RoboDK station: Estacion_Paletizado.rdk

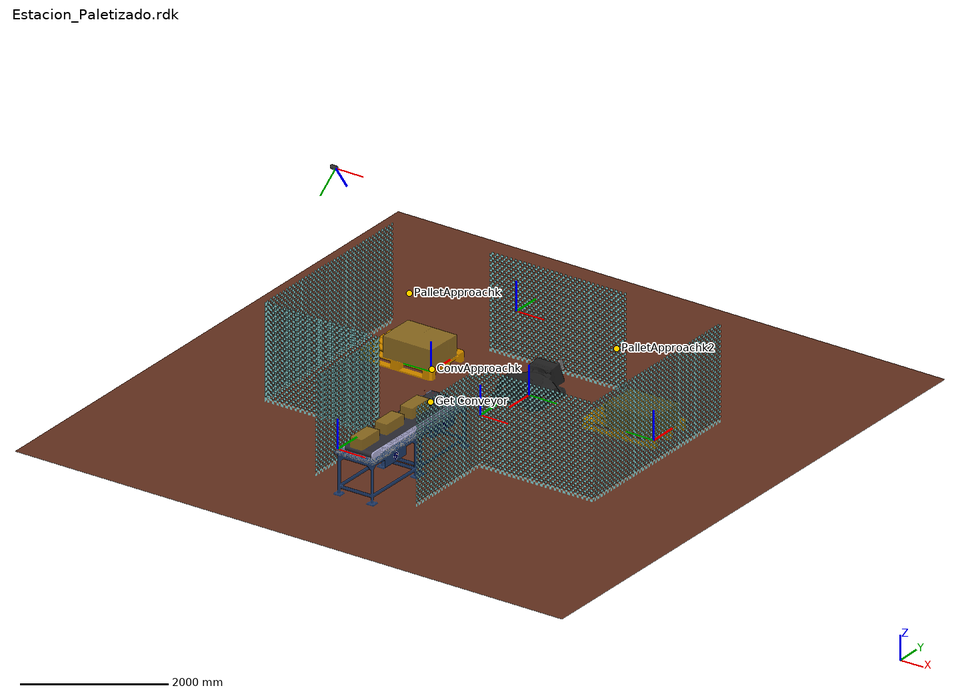
[picture v0: the station drawn from its stored meshes, robots at their saved joint values, targets as dots, program paths as lines]
Station Estacion_Paletizado (saved by RoboDK 5.3.2). Poses are relative to the parent item; angles as X-Y-Z fixed-axis rotations.
Station parameters (name, value as stored): SizeBox, 200, 400, 160, SizePallet, 3,2,2, ConvSpeed, 100.0, SENSOR, 0, parts/min, 2.5, BOX, 84, NBOXP, 12.0, EPALLETE, 1,1, FOTO, 0
  - frame Mundo at (700, 2520, -620) mm
    - object Floor at (0, 0, 0) mm, size 9000 x 9000 x 0 mm, geometry from Floor.sld
    - object Plane 1m x 1m grid at (-725, -2080, 760) mm, rotated rx 0 ry 90 rz 0 deg, size 1500 x 1500 x 0.8 mm, geometry from plane_1m_grid.sld
    - object Plane 1m x 1m grid at (-1850, -1340, 760) mm, rotated rx 0 ry 90 rz 90 deg, size 1500 x 1500 x 0.8 mm, geometry from plane_1m_grid.sld
    - object Plane 1m x 1m grid at (-2600, 910, 750) mm, rotated rx 0 ry 90 rz 0 deg, size 1500 x 1500 x 0.8 mm, geometry from plane_1m_grid.sld
    - object Plane 1m x 1m grid at (-1475, -1340, 760) mm, rotated rx 0 ry 90 rz 90 deg, size 1500 x 1500 x 0.8 mm, geometry from plane_1m_grid.sld
    - object Plane 1m x 1m grid at (-265, 1670, 760) mm, rotated rx 0 ry 90 rz -90 deg, size 1500 x 1500 x 0.8 mm, geometry from plane_1m_grid.sld
    - object Plane 1m x 1m grid at (485, 1670, 760) mm, rotated rx 0 ry 90 rz -90 deg, size 1500 x 1500 x 0.8 mm, geometry from plane_1m_grid.sld
    - object Plane 1m x 1m grid at (2795, 910, 760) mm, rotated rx 0 ry 90 rz -180 deg, size 1500 x 1500 x 0.8 mm, geometry from plane_1m_grid.sld
    - object Plane 1m x 1m grid at (2795, -590, 760) mm, rotated rx 0 ry 90 rz -180 deg, size 1500 x 1500 x 0.8 mm, geometry from plane_1m_grid.sld
    - object Plane 1m x 1m grid at (2040, -1340, 760) mm, rotated rx 0 ry 90 rz 90 deg, size 1500 x 1500 x 0.8 mm, geometry from plane_1m_grid.sld
    - object Plane 1m x 1m grid at (-2600, -590, 760) mm, rotated rx 0 ry 90 rz 0 deg, size 1500 x 1500 x 0.8 mm, geometry from plane_1m_grid.sld
    - object Plane 1m x 1m grid at (1665, -1340, 760) mm, rotated rx 0 ry 90 rz 90 deg, size 1500 x 1500 x 0.8 mm, geometry from plane_1m_grid.sld
    - object Plane 1m x 1m grid at (925, -2080, 760) mm, rotated rx 0 ry 90 rz 0 deg, size 1500 x 1500 x 0.8 mm, geometry from plane_1m_grid.sld
    - object Table 1400x800x800 at (110, -1140, 645) mm, rotated rx 0 ry 0 rz -90 deg, size 1138.7 x 657.6 x 641.5 mm, geometry from Table-1400mmx800mmx800mm.sld
    - object Table 1400x800x800 at (110, -2280, 645) mm, rotated rx 0 ry 0 rz -90 deg, size 1138.7 x 657.6 x 641.5 mm, geometry from Table-1400mmx800mmx800mm.sld
  - frame KR Base at (900, 3380, -610) mm, rotated rx 0 ry 0 rz -90 deg
    - robot KR (model KUKA KR 120 R3200 PA): 4 axes, payload 120 kg, reach 3195 mm, repeatability 0.06 mm, weight 1075 kg
        joint limits [-185, -140, 0, -350] to [185, -5, 155, 350]; home [0, -100.15, 95.16, -180.59]; saved at [80.379, -89.016, 111.792, -188.281]
      - tool GripperK, TCP at (0, 0, 80) mm, rotated rx 0 ry 0 rz 90 deg, size 461.9 x 92.4 x 220 mm, geometry from test.iges
      - tool TCPK, TCP at (0, 0, 160) mm, rotated rx 0 ry 0 rz 90 deg
    - target ConvApproachk (joint target) at (2164.54, -72.94, 1237.21) mm, rotated rx -180 ry 0 rz -90.59 deg; joints [1.93, -73.65, 92.328, -178.66, 0, 0] of KR
    - target PalletApproachk (joint target) at (297.16, -1753.05, 1156.5) mm, rotated rx 180 ry 0 rz -178.66 deg; joints [80.379, -89.016, 111.792, -188.281, 0, 0] of KR
    - target PalletApproachk2 (joint target) at (316.59, 1666.46, 1294.36) mm, rotated rx 180 ry 0 rz -180 deg; joints [-79.243, -94.763, 109.774, 10.757] of KR
    - frame PalletK2 at (419.96, 2346.44, 151.5) mm, rotated rx 0 ry 0 rz 180 deg
      - object EuropalletK at (0, 0, 0) mm, size 800 x 144 x 1200 mm, geometry from User Library-Europallet.igs
      - object Part at (100.16, 200.94, 79.97) mm, rotated rx 0 ry 0 rz -180 deg, size 200 x 400 x 160 mm, geometry from box.sld
      - object Part at (300.16, 202.94, 79.97) mm, rotated rx 0 ry 0 rz -180 deg, size 200 x 400 x 160 mm, geometry from box.sld
      - object Part at (500.16, 199.94, 79.97) mm, rotated rx 0 ry 0 rz 180 deg, size 200 x 400 x 160 mm, geometry from box.sld
      - object Part at (100.16, 579.94, 79.97) mm, rotated rx 0 ry 0 rz 180 deg, size 200 x 400 x 160 mm, geometry from box.sld
      - object Part at (300.16, 601.94, 79.97) mm, rotated rx 0 ry 0 rz 180 deg, size 200 x 400 x 160 mm, geometry from box.sld
      - object Part at (500.16, 600.94, 79.97) mm, rotated rx 0 ry 0 rz -180 deg, size 200 x 400 x 160 mm, geometry from box.sld
      - object Part at (100.16, 199.94, 239.97) mm, rotated rx 0 ry 0 rz 180 deg, size 200 x 400 x 160 mm, geometry from box.sld
      - object Part at (300.16, 202.94, 239.97) mm, rotated rx 0 ry 0 rz 180 deg, size 200 x 400 x 160 mm, geometry from box.sld
      - object Part at (500.16, 202.94, 239.97) mm, rotated rx 0 ry 0 rz -180 deg, size 200 x 400 x 160 mm, geometry from box.sld
      - object Part at (100.16, 602.94, 239.97) mm, rotated rx 0 ry 0 rz -180 deg, size 200 x 400 x 160 mm, geometry from box.sld
      - object Part at (300.16, 607.94, 239.97) mm, rotated rx 0 ry 0 rz -180 deg, size 200 x 400 x 160 mm, geometry from box.sld
      - object Part at (500.16, 598.94, 239.97) mm, rotated rx 0 ry 0 rz 180 deg, size 200 x 400 x 160 mm, geometry from box.sld
    - frame PalletK at (419.96, -1313.56, 151.5) mm, rotated rx 0 ry 0 rz 180 deg
      - object EuropalletK at (0, 0, 0) mm, size 800 x 144 x 1200 mm, geometry from User Library-Europallet.igs
      - object Part at (100.16, 203.94, 79.97) mm, rotated rx 0 ry 0 rz 180 deg, size 200 x 400 x 160 mm, geometry from box.sld
      - object Part at (300.16, 202.94, 79.97) mm, rotated rx 0 ry 0 rz -180 deg, size 200 x 400 x 160 mm, geometry from box.sld
      - object Part at (500.16, 202.94, 79.97) mm, rotated rx 0 ry 0 rz 180 deg, size 200 x 400 x 160 mm, geometry from box.sld
      - object Part at (100.16, 596.94, 79.97) mm, rotated rx 0 ry 0 rz -180 deg, size 200 x 400 x 160 mm, geometry from box.sld
      - object Part at (300.16, 602.94, 79.97) mm, rotated rx 0 ry 0 rz -180 deg, size 200 x 400 x 160 mm, geometry from box.sld
      - object Part at (500.16, 603.94, 79.97) mm, rotated rx 0 ry 0 rz 180 deg, size 200 x 400 x 160 mm, geometry from box.sld
      - object Part at (100.16, 201.94, 239.97) mm, rotated rx 0 ry 0 rz -180 deg, size 200 x 400 x 160 mm, geometry from box.sld
      - object Part at (300.16, 201.94, 239.97) mm, rotated rx 0 ry 0 rz 180 deg, size 200 x 400 x 160 mm, geometry from box.sld
      - object Part at (500.16, 194.94, 239.97) mm, rotated rx 0 ry 0 rz 180 deg, size 200 x 400 x 160 mm, geometry from box.sld
      - object Part at (100.16, 596.94, 239.97) mm, rotated rx 0 ry 0 rz 180 deg, size 200 x 400 x 160 mm, geometry from box.sld
      - object Part at (300.16, 602.94, 239.97) mm, rotated rx 0 ry 0 rz 180 deg, size 200 x 400 x 160 mm, geometry from box.sld
      - object Part at (500.16, 599.94, 239.97) mm, rotated rx 0 ry 0 rz -180 deg, size 200 x 400 x 160 mm, geometry from box.sld
  - frame ConveyorReference at (597.23, -679.82, 119.18) mm
    - robot Conveyor Belt: 1 axes
        modified DH rows (alpha deg, a mm, theta deg, d mm): 0, 0, 0, 0 linear
        base shift (440, 200, 0) mm, rotated rx 0 ry 90 rz 90 deg
        joint limits [-500000] to [500000]; home [0]; saved at [50536]
      - frame MovingRef at (0, 0, 0) mm
        - object Part at (-49217, 240, 80) mm, rotated rx 0 ry 0 rz -90 deg, size 200 x 400 x 160 mm, geometry from box.sld
        - object Part at (-49811, 240, 80) mm, rotated rx 0 ry 0 rz -90 deg, size 200 x 400 x 160 mm, geometry from box.sld
        - object Part at (-50391, 240, 80) mm, rotated rx 0 ry 0 rz -90 deg, size 200 x 400 x 160 mm, geometry from box.sld
    - object box100mm at (200, 300, 0) mm, size 100 x 100 x 100 mm, geometry from box.sld
    - object Sensor SICK WL4S at (551.19, 2078.29, 24.16) mm, rotated rx 90 ry 0 rz 180 deg, size 683.3 x 45.2 x 12.5 mm, geometry from SICK WL4S-3P1330-Order no.1042068 (1).stp
      - Python program SensorActivate (listed below)
    - target Get Conveyor (Cartesian target) at (200.16, 1899.94, 0.03) mm, rotated rx -180 ry 0 rz -180 deg; joints [2.72, -64.765, 103.115, -177.28, 0, 0] of KR
  - frame Camera Reference at (780, -980, 4500) mm, rotated rx -145 ry 0 rz 0 deg
    - object SICK VSPP-5f2113 at (0, 0, 0) mm, size 53 x 116 x 38 mm, geometry from Cam2D_SICK_VSPP_5F2113.sld
  - Python program SetSimulationParams (listed below)
  - Python program BorradoA (listed below)
  - Python program BorradoB (listed below)
  - Python program AddPart (listed below)
  - Python program InputParts (listed below)
  - Python program RobotPackParts (listed below)
  - Python program Telegram (listed below)
  - Python program Camara (listed below)
  - program MainSimulation (5 instructions, listed below)
  - frame Fajardo_Jacho at (0, 4380, 0) mm

--- Python program SensorActivate ---
# Type help("robolink") or help("robodk") for more information
# Press F5 to run the script
# Note: you do not need to keep a copy of this file, your python script is saved with the station
from robolink import *    # API to communicate with RoboDK
from robodk import *      # basic matrix operations
RDK = Robolink()

# This script allows to simulate a laser sensor
# that detect the presence of a part in a plane,
# such as a part crossing a laser sensor in a
# conveyor belt

# Use a target from the station as a reference plane:
SENSOR_NAME = 'Sensor SICK WL4S'
SENSOR_VARIABLE = 'SENSOR'

# Look for parts with the keyword "Part"
OBJECTS_REFERENCE = 'MovingRef'
moving_ref = RDK.Item(OBJECTS_REFERENCE, ITEM_TYPE_FRAME)

# Update status every 1 ms
RECHECK_PERIOD = 0.001

# Get the sensor and the detection plane
SENSOR = RDK.Item(SENSOR_NAME, ITEM_TYPE_OBJECT)

# Start delayed as some parts may be deleted
pause(2)

# Loop forever to detect parts
detected_status = -1
while True:
    detected = 0
    for obj in moving_ref.Childs():
        # check if an object has the part keyword and is detected by the laser
        if SENSOR.Collision(obj) > 0:
            detected = 1
            break

    # update the current status of the sensor
    if detected_status != detected:
        detected_status = detected
        RDK.setParam(SENSOR_VARIABLE, detected_status)
        print('Object detected status --> %i' % detected_status)

    ESTADOS_PALLET      = RDK.getParam('EPALLETE')
    ESTADOS_PALLET_AB   = [int(x.replace(' ','')) for x in ESTADOS_PALLET.split(',')]
    numero_disponible   = ESTADOS_PALLET_AB[0] + ESTADOS_PALLET_AB[1]

    if numero_disponible == 2:
        # Se detiene el sensor hasta que haya palletes disponibles
        while numero_disponible == 2:
            ESTADOS_PALLET      = RDK.getParam('EPALLETE')
            ESTADOS_PALLET_AB   = [int(x.replace(' ','')) for x in ESTADOS_PALLET.split(',')]
            numero_disponible   = ESTADOS_PALLET_AB[0] + ESTADOS_PALLET_AB[1]
        pause(2)
    # Wait some time...
    pause(RECHECK_PERIOD)

--- Python program SetSimulationParams ---
# Type help("robolink") or help("robodk") for more information
# Press F5 to run the script
# Note: you do not need to keep a copy of this file, your python script is saved with the station
from robolink import *    # API to communicate with RoboDK
from robodk import *      # basic matrix operations

RDK = Robolink()

# Parametros creados en la estacion de trabajo
PARAM_SIZE_BOX = 'SizeBox'
PARAM_SIZE_PALLET = 'SizePallet'
PARAM_CONV_SPEED_MM = 'ConvSpeed'
PARAM_PARTS_X_MINUTE = 'parts/min'

#Valores de los parametros creados en la estacion de trabajo
size_box = RDK.getParam(PARAM_SIZE_BOX)
size_pallet = RDK.getParam(PARAM_SIZE_PALLET)
conv_speed = RDK.getParam(PARAM_CONV_SPEED_MM)
parts_x_minute = RDK.getParam(PARAM_PARTS_X_MINUTE)

# ------------------------------------------------------------
size_box_input = mbox('Enter the size of the box in mm [L,W,H]', entry=size_box)
if size_box_input:
    RDK.setParam(PARAM_SIZE_BOX, size_box_input)
else:
    quit()

# ------------------------------------------------------------
size_pallet_input = mbox('Enter the size of the pallet', entry=size_pallet)
if size_pallet_input:
    RDK.setParam(PARAM_SIZE_PALLET, size_pallet_input)
else:
    quit()


# ------------------------------------------------------------
parts_x_minute_entry = mbox('Enter the number of parts per minute', entry=parts_x_minute)
if parts_x_minute_entry:
    RDK.setParam(PARAM_PARTS_X_MINUTE, parts_x_minute_entry)
else:
    quit()

# ------------------------------------------------------------
conv_speed_input = mbox('Enter the speed of the conveyor in mm/s', entry=conv_speed)
if conv_speed_input:
    RDK.setParam(PARAM_CONV_SPEED_MM, conv_speed_input)
    conv_speed = float(conv_speed_input)
    conv = RDK.Item('Conveyor Belt', ITEM_TYPE_ROBOT)
    conv.setSpeed(conv_speed)

else:
    quit()

--- Python program BorradoA ---
# Type help("robolink") or help("robodk") for more information
# Press F5 to run the script
# Documentation: https://robodk.com/doc/en/RoboDK-API.html
# Reference:     https://robodk.com/doc/en/PythonAPI/index.html
# Note: It is not required to keep a copy of this file, your python script is saved with the station
from robolink import *    # RoboDK API
from robodk import *      # Robot toolbox
RDK = Robolink()

# Variable con la referencia del pallete a borrar
pallete_ref = RDK.Item('PalletK', ITEM_TYPE_FRAME)

#Eliminar las cajas del PalleteA
for obj in pallete_ref.Childs():
    if obj.Name().startswith("Part"):
        obj.Delete()

# Actualizar el estado de palleteA en el parametro EPALLETE
estado_pallete = RDK.getParam('EPALLETE')
l = list(estado_pallete) #El parametro es un string
l[0] = '0'
estado_pallete = "".join(l)
RDK.setParam('EPALLETE', estado_pallete)

--- Python program BorradoB ---
# Type help("robolink") or help("robodk") for more information
# Press F5 to run the script
# Documentation: https://robodk.com/doc/en/RoboDK-API.html
# Reference:     https://robodk.com/doc/en/PythonAPI/index.html
# Note: It is not required to keep a copy of this file, your python script is saved with the station
from robolink import *    # RoboDK API
from robodk import *      # Robot toolbox
RDK = Robolink()

# Variable con la referencia del pallete a borrar
pallete_ref = RDK.Item('PalletK2', ITEM_TYPE_FRAME)

#Eliminar las cqjas del PalleteB
for obj in pallete_ref.Childs():
    if obj.Name().startswith("Part"):
        obj.Delete()

# Actualizar el estado de palleteB en el parametro EPALLETE
estado_pallete = RDK.getParam('EPALLETE')
l = list(estado_pallete) #El parametro es un string
l[2] = '0'
estado_pallete = "".join(l)
RDK.setParam('EPALLETE', estado_pallete)

--- Python program AddPart ---
# Type help("robolink") or help("robodk") for more information
# Press F5 to run the script
# Note: you do not need to keep a copy of this file, your python script is saved with the station
from robolink import *    # API to communicate with RoboDK
from robodk import *      # basic matrix operations
import random
RDK = Robolink()

#Variables con nombre de objeto y referencia a usar
PART_NAME       = 'box100mm'
CONVEYOR_REF    = 'MovingRef'

#Valores de las dimensiones de la caja
SIZE_BOX = RDK.getParam('SizeBox')
SIZE_BOX_XYZ = [float(x.replace(' ','')) for x in SIZE_BOX.split(',')]
[SIZE_BOX_X, SIZE_BOX_Y, SIZE_BOX_Z] = SIZE_BOX_XYZ

# Creacion de nueva caja en la banda
part = RDK.Item(PART_NAME, ITEM_TYPE_OBJECT)
conveyor_ref = RDK.Item(CONVEYOR_REF, ITEM_TYPE_FRAME) #Referencia movil de la banda transportadora
part_pos = part.PoseAbs() # Posicion absoluta de la caja de referencia
part.Copy()
newpart = conveyor_ref.Paste()
newpart.setPoseAbs(part_pos*transl(0,0,SIZE_BOX_Z/2)) #Posicionando la nueva caja teniendo en cuenta su referencia central.
newpart.setName('Part') # Se crea una caja para el palleteA
newpart.Scale([SIZE_BOX_X/100, SIZE_BOX_Y/100, SIZE_BOX_Z/100]) #Escala con respecto al objeto de referencia (100mm cube)
newpart.Recolor([0.678, 0.529, 0.2, 1]) #set RGBA color
newpart.setVisible(True, False) #make item visible but hide the reference frame

--- Python program InputParts ---
# Type help("robolink") or help("robodk") for more information
# Press F5 to run the script
# Note: you do not need to keep a copy of this file, your python script is saved with the station
from robolink import *    # API to communicate with RoboDK
from robodk import *      # basic matrix operations

# Use RoboDK API as RDK
RDK = Robolink()

# Parametros de la estacion
PARAM_PARTS_X_MINUTE = 'parts/min'
PARAM_NUMERO_BOX_PALLETE = 'NBOXP'
PARAM_ESTADO_PALLETE = 'EPALLETE'

# Establecer en 0 el estado de los pallete A y B
RDK.setParam(PARAM_ESTADO_PALLETE, '0,0')

# Establecer el numero indicador de cajas por Pallete
SIZE_PALLET = RDK.getParam('SizePallet')
SIZE_PALLET_XYZ = [float(x.replace(' ','')) for x in SIZE_PALLET.split(',')]
numero_box_pallete = SIZE_PALLET_XYZ[0]*SIZE_PALLET_XYZ[1]*SIZE_PALLET_XYZ[2]
RDK.setParam(PARAM_NUMERO_BOX_PALLETE, numero_box_pallete)

# turn off rendering (much faster when setting up the station)
#RDK.Render(False)

# Eliminar todas las cajas previamente simuladas
all_objects     = RDK.ItemList(ITEM_TYPE_OBJECT, False)
for item in all_objects:
    if item.Name().startswith("Part"):
        item.Delete()

# Turn on rendering
#RDK.Render(True)

# Valor de la cantidad de cajas por minuto
parts_x_minute = RDK.getParam(PARAM_PARTS_X_MINUTE)

# Seleccion del codigo de AddPart
add_part = RDK.Item('AddPart', ITEM_TYPE_PROGRAM_PYTHON)

# Movimiento de la banda transportadora
conv = RDK.Item('Conveyor Belt', ITEM_TYPE_ROBOT)
conv.setJoints([0]) # Establecer en cero
conv.MoveJ([99999], False) # Mover hasta el maximo valor permitido.

# Temporizador para creacion de cajas
SECONDS_X_PART = 60.0 / parts_x_minute #Tiempo por cada caja
tic() # Marcar inicio de cconteo
timer_last = toc() # Tiempo transcurrido desde el inicio del conteo
simulation_time = SECONDS_X_PART
while True:

    # Numero indicador de disponibilidad de pallete
    ESTADOS_PALLET      = RDK.getParam(PARAM_ESTADO_PALLETE)
    ESTADOS_PALLET_AB   = [int(x.replace(' ','')) for x in ESTADOS_PALLET.split(',')]
    numero_disponible   = ESTADOS_PALLET_AB[0] + ESTADOS_PALLET_AB[1]

    # Creacion de la nueva caja
    timer = toc()
    simulation_time = simulation_time + (timer - timer_last) * RDK.SimulationSpeed()
    timer_last = timer
    if simulation_time >= SECONDS_X_PART and numero_disponible != 2: # Se crea mas cajas siempre que haya disponibles un pallete
        simulation_time = simulation_time - SECONDS_X_PART
        add_part.RunProgram()
    if numero_disponible == 2: # No hay disponible pallete
        conv.Stop()
        while numero_disponible == 2: #Espera hasta este disponible el palleteA
            ESTADOS_PALLET      = RDK.getParam(PARAM_ESTADO_PALLETE)
            ESTADOS_PALLET_AB   = [int(x.replace(' ','')) for x in ESTADOS_PALLET.split(',')]
            numero_disponible   = ESTADOS_PALLET_AB[0] + ESTADOS_PALLET_AB[1]
        conv.MoveJ([99999], False)
        tic() # Se reinicia la cuenta para las cajas
        timer_last = toc()
        simulation_time = 0

    pause(0.01)

--- Python program RobotPackParts ---
# Type help("robolink") or help("robodk") for more information
# Press F5 to run the script
# Note: you do not need to keep a copy of this file, your python script is saved with the station
from robolink import *    # API to communicate with RoboDK
from robodk import *      # basic matrix operations

# Use RoboDK API as RL
RDK = Robolink()

# define default approach distance
APPROACH = 100

# Parametros de la estacion
SENSOR_VARIABLE = 'SENSOR'
PARAM_ESTADO_PALLETE = 'EPALLETE'
RDK.setParam(PARAM_ESTADO_PALLETE, '0,0')
ESTADOS_PALLET      = RDK.getParam(PARAM_ESTADO_PALLETE)

# gather robot, tool and reference frames from the station
robot               = RDK.Item('KR', ITEM_TYPE_ROBOT)
tool                = RDK.Item('GripperK', ITEM_TYPE_TOOL)
tool_tcp            = RDK.Item('TCPK', ITEM_TYPE_TOOL)

frame_palletA        = RDK.Item('PalletK', ITEM_TYPE_FRAME)
frame_palletB       = RDK.Item('PalletK2', ITEM_TYPE_FRAME)
frame_conv          = RDK.Item('ConveyorReference', ITEM_TYPE_FRAME)
frame_conv_moving   = RDK.Item('MovingRef', ITEM_TYPE_FRAME)

# gather targets
target_pallet_safeA  = RDK.Item('PalletApproachk', ITEM_TYPE_TARGET)
target_pallet_safeB = RDK.Item('PalletApproachk2', ITEM_TYPE_TARGET)
target_conv_safe    = RDK.Item('ConvApproachk', ITEM_TYPE_TARGET)
target_conv         = RDK.Item('Get Conveyor', ITEM_TYPE_TARGET)

# Reinicio de la cuenta de las cajas totales paletizadas
COUNT_BOX = 0

# get variable parameters
SIZE_BOX = RDK.getParam('SizeBox')
SIZE_PALLET = RDK.getParam('SizePallet')
SIZE_BOX_XYZ = [float(x.replace(' ','')) for x in SIZE_BOX.split(',')]
SIZE_PALLET_XYZ = [float(x.replace(' ','')) for x in SIZE_PALLET.split(',')]
SIZE_BOX_Z = SIZE_BOX_XYZ[2] # the height of the boxes is important to take into account when approaching the positions

def box_calc(size_xyz, pallet_xyz):
    """Calculates a list of points to store parts in a pallet"""
    [size_x, size_y, size_z] = size_xyz
    [pallet_x, pallet_y, pallet_z] = pallet_xyz
    xyz_list = []
    for h in range(int(pallet_z)):
        for j in range(int(pallet_y)):
            for i in range(int(pallet_x)):
                xyz_list = xyz_list + [[(i+0.5)*size_x, (j+0.5)*size_y, (h+0.5)*size_z]]
    return xyz_list

def TCP_On(toolitem):
    """Attaches the closest object to the toolitem Htool pose,
    It will also output appropriate function calls on the generated robot program (call to TCP_On)"""
    toolitem.AttachClosest()
    toolitem.RDK().RunMessage('Set air valve on')
    toolitem.RDK().RunProgram('TCP_On()')

def TCP_Off(toolitem, itemleave=0):
    """Detaches the closest object attached to the toolitem Htool pose,
    It will also output appropriate function calls on the generated robot program (call to TCP_Off)"""
    #toolitem.DetachClosest(itemleave)
    toolitem.DetachAll(itemleave)
    toolitem.RDK().RunMessage('Set air valve off')
    toolitem.RDK().RunProgram('TCP_Off()')

# calculate an array of positions to get/store the parts
parts_positions = box_calc(SIZE_BOX_XYZ, SIZE_PALLET_XYZ)

# Calculate a new TCP that takes into account the size of the part (targets are set to the center of the box)
tool_xyzrpw = tool.PoseTool()*transl(0,0,SIZE_BOX_Z/2)
tool_tcp.setPoseTool(tool_xyzrpw)
#tool_tcp = robot.AddTool(tool_xyzrpw, 'TCP')

# ---------------------------------------------------------------------------------
# -------------------------- PROGRAM START ----------------------------------------

def WaitSensor():
    if RDK.RunMode() == RUNMODE_SIMULATE:
        # Simulate the sensor by waiting for the SENSOR status to turn to 1 (object present)
        while RDK.getParam(SENSOR_VARIABLE) == 0:
            pause(0.001)
    else:
        RDK.RunProgram('WaitSensor')
    print("Part detected")

P = -1 # Variable indicadora del pallete a llenar
robot.setTool(tool_tcp)
nparts = len(parts_positions)
while True:
    # Numero indicador de disponibilidad de palletes
    ESTADOS_PALLET_AB   = [int(x.replace(' ','')) for x in ESTADOS_PALLET.split(',')]
    numero_disponible   = ESTADOS_PALLET_AB[0] + ESTADOS_PALLET_AB[1]

    if numero_disponible == 2:
        # Se detiene el brazo robotico hasta que haya palletes disponibles
        while numero_disponible == 2:
            ESTADOS_PALLET      = RDK.getParam(PARAM_ESTADO_PALLETE)
            ESTADOS_PALLET_AB   = [int(x.replace(' ','')) for x in ESTADOS_PALLET.split(',')]
            numero_disponible   = ESTADOS_PALLET_AB[0] + ESTADOS_PALLET_AB[1]
    #Establecer la referencia y el target del pallete
    if ESTADOS_PALLET_AB[0] == 0:
        P = 1
        frame_pallet = frame_palletA
        target_pallet_safe = target_pallet_safeA
    elif ESTADOS_PALLET_AB[1] == 0:
        P = 2
        frame_pallet = frame_palletB
        target_pallet_safe = target_pallet_safeB

    i = 0
    while i < nparts:
        # ----------- place the box i on the convegor ------
        # approach to the conveyor
        robot.setFrame(frame_conv)
        target_conv_pose = target_conv.Pose()*transl(0,0,-SIZE_BOX_Z/2)
        target_conv_app = target_conv_pose*transl(0,0,-APPROACH)
        robot.MoveJ(target_conv_safe)
        robot.MoveJ(target_conv_app)
        WaitSensor()
        robot.MoveL(target_conv_pose)
        TCP_On(tool) # detach an place the object in the moving reference frame of the conveyor
        robot.MoveL(target_conv_app)
        robot.MoveJ(target_conv_safe)

        # ----------- take a part from the conveyor ------
        # get the xyz position of part i
        robot.setFrame(frame_pallet)
        part_position_i = parts_positions[i]
        target_i = transl(part_position_i)*rotx(pi)
        target_i_app = target_i * transl(0,0,-(APPROACH+SIZE_BOX_Z))
        # approach to the pallet
        robot.MoveJ(target_pallet_safe)
        # get the box i
        robot.MoveJ(target_i_app)
        robot.MoveL(target_i)
        TCP_Off(tool, frame_pallet) # attach the closest part
        robot.MoveL(target_i_app)
        robot.MoveJ(target_pallet_safe)
        COUNT_BOX +=1 # Aumenta la cuenta cuando deja una caja
        RDK.setParam('BOX', COUNT_BOX)
        i = i + 1

    # Cambio del estado de los pallete
    ESTADOS_PALLET      = RDK.getParam(PARAM_ESTADO_PALLETE)
    if P == 1:
        l = list(ESTADOS_PALLET)
        l[0] = '1'
        ESTADOS_PALLET = "".join(l)
    else:
        l = list(ESTADOS_PALLET)
        l[2] = '1'
        ESTADOS_PALLET = "".join(l)
    RDK.setParam('EPALLETE', ESTADOS_PALLET)

--- Python program Telegram ---
#!/usr/bin/env python
# pylint: disable=C0116,W0613
# This program is dedicated to the public domain under the CC0 license.

import logging

from telegram import Update, ForceReply
from telegram.ext import Updater, CommandHandler, MessageHandler, Filters, CallbackContext
from telegram import ChatAction

# Enable logging
logging.basicConfig(
    format='%(asctime)s - %(name)s - %(levelname)s - %(message)s', level=logging.INFO
)

logger = logging.getLogger(__name__)


from robolink import *    # RoboDK API
from robodk import *      # Robot toolbox

RDK = Robolink()
FOTO_ESTACION = 'FOTO' # Parametro que indica si se debe tomar una foto
path_rdk = RDK.getParam('PATH_OPENSTATION')# Parametro con la direccion de la foto
file_name = '/estacion.jpg'# Parametro con el nombre de la foto

# Definiendo los comandos de telegram
def start(update: Update, context: CallbackContext) -> None:
    user = update.effective_user
    update.message.reply_markdown_v2( #Funcion para enviar un mensaje con el nombre del usuario.
        fr'Hola {user.mention_markdown_v2()}\!',
        reply_markup=ForceReply(selective=True),
    )
    update.message.reply_text('En esta aplicacion podras consultar el estado de la estacion de paletizado, usa el comando /help para conocer las funciones')

def help_command(update: Update, context: CallbackContext) -> None:
    update.message.reply_text('Las funciones que se pueden usar son:') # Funcion para enviar un mensaje de texto al usuario
    update.message.reply_text('/help -> Te ayuda a conocer la funciones existentes')
    update.message.reply_text('/box -> Te indica la cantidas de cajas paletizadas')
    update.message.reply_text('/pallete -> Te indica la cantidad de palletes llenos')
    update.message.reply_text('/Epallete -> Te indica el estado de los palletes de la estacion')
    update.message.reply_text('/foto -> Te envia una foto de la estacion')

def echo(update: Update, context: CallbackContext) -> None:
    update.message.reply_text('Por favor, ingrese un comando conocido, o de clic en -> /help')

def box(update: Update, context: CallbackContext) -> None:
    cantidad_cajas = RDK.getParam('BOX') # Parametro con el valor de cajas totales paletizadas
    update.message.reply_text('La cantidad de cajas paletizadas es de ' + str(cantidad_cajas))

def pallete(update: Update, context: CallbackContext) -> None:
    cantidad_cajas = int(RDK.getParam('BOX')) # Parametro con el valor de cajas totales paletizadas
    numero_box_pallete = int(RDK.getParam('NBOXP')) #Parametro con la cantidad de cajas por palleto
    cantidad_pallete = cantidad_cajas//numero_box_pallete # Numero de palletes enteros realizados
    update.message.reply_text('La cantidad de palletes terminados es de ' + str(cantidad_pallete))

def Epallete(update: Update, context: CallbackContext) -> None:
    estado_pallete      = RDK.getParam('EPALLETE') #Parametro con el estado de los palletes
    estados_pallete_AB   = [int(x.replace(' ','')) for x in estado_pallete.split(',')]
    # Asignacion de vacio o lleno al mensaje sobre el estado de cada pallete
    if estados_pallete_AB[0] == 0 :
        palleteA = 'vacio o llenando'
    else:
        palleteA = 'lleno'
    if estados_pallete_AB[1] == 0:
        palleteB = 'vacio o llenando'
    else:
        palleteB = 'lleno'

    # Determinar estructura del mensaje segun el estado de los palletes
    if estados_pallete_AB == [1,1]:
        update.message.reply_text('Los dos palletes se encuentran llenos, el proceso esta detenido' )
    else:
        update.message.reply_text('El palleteA esta ' + str(palleteA))
        update.message.reply_text('El palleteB esta ' + str(palleteB))

def foto(chat):
    chat.send_action(action=ChatAction.UPLOAD_PHOTO,timeout=None) #Accion de que se esta enviando una foto
    pause(0.1)
    chat.send_photo(photo = open(path_rdk+file_name,'rb')) # Se envia la foto que sera buscada en la direccion establecida
    RDK.setParam(FOTO_ESTACION,'0') # Actualizacion de parametro que indica cuando tomar una foto

def chat(update: Update, context: CallbackContext) -> None:
    RDK.setParam(FOTO_ESTACION,'1') # Actualizacion de parametro que indica cuando tomar una foto
    chat = update.message.chat #Datos de chat de la persona que escribe
    foto(chat) # Funcion para enviar la foto

def main() -> None:
    """Start the bot."""
    # Create the Updater and pass it your bot's token.
    updater = Updater("5062967228:AAGSuI74jk8Jqe0g8b1kAKCBIIlwF6qlM4A")

    # Get the dispatcher to register handlers
    dispatcher = updater.dispatcher

    # on different commands - answer in Telegram
    dispatcher.add_handler(CommandHandler("start", start))
    dispatcher.add_handler(CommandHandler("help", help_command))
    dispatcher.add_handler(CommandHandler("box", box))
    dispatcher.add_handler(CommandHandler("pallete", pallete))
    dispatcher.add_handler(CommandHandler("Epallete", Epallete))
    dispatcher.add_handler(CommandHandler("foto", chat))

    # on non command i.e message - echo the message on Telegram
    dispatcher.add_handler(MessageHandler(Filters.text & ~Filters.command, echo))

    # Start the Bot
    updater.start_polling()
    # Run the bot until you press Ctrl-C or the process receives SIGINT,
    # SIGTERM or SIGABRT. This should be used most of the time, since
    # start_polling() is non-blocking and will stop the bot gracefully.
    updater.idle()


if __name__ == '__main__':
    main()

--- Python program Camara ---
# Type help("robolink") or help("robodk") for more information
# Press F5 to run the script
# Note: you do not need to keep a copy of this file, your python script is saved with the station
from robolink import *    # API to communicate with RoboDK
from robodk import *      # basic matrix operations
RDK = Robolink()

#Parametro que indica cuando tomar una foto
FOTO_ESTACION = 'FOTO'

#Direccion y nombre de la foto
path_rdk = RDK.getParam('PATH_OPENSTATION')
file_name = '/estacion.jpg'

while(1):
    ref_cam = RDK.Item('Camera Reference',ITEM_TYPE_FRAME)
    ref_cam.setVisible(False)

    tomar_foto = int(RDK.getParam(FOTO_ESTACION)) # Indicador para tomar la foto
    while tomar_foto == 0: # No tomara la foto mientras se indique 0
        tomar_foto = int(RDK.getParam(FOTO_ESTACION))
        pause(0.001)
    #Parametros, toma y guardado de la foto.
    cam_id = RDK.Cam2D_Add(ref_cam, 'FOCAL_LENGHT=6 FOV=32 FAR_LENGHT=10000 SIZE=1024x768 BG_COLOR=black LIGHT_AMBIENT=white LIGHT_DIFFUSE=black LIGHT_SPECULAR=white')
    RDK.Cam2D_Snapshot((path_rdk+file_name), cam_id)
    RDK.Cam2D_Close(cam_id)
    cam_id.Delete()

    while tomar_foto == 1: #No tomara otra foto hasta que se resetee el indicador.
        tomar_foto = int(RDK.getParam(FOTO_ESTACION))
        pause(0.001)

--- program MainSimulation ---
  Run RobotPackParts
  Run SensorActivate
  Run InputParts
  Ejecutar Camara
  Ejecutar Telegram
